FUNCTION_BLOCK SWITCHsim (* Service Interface Function Block Type *)
  (* Standard: 61499-2 *)
  (* Version 1.0, 2020-01-13, badger *)
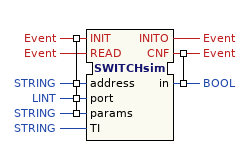
  EVENT_INPUT
    INIT WITH address, port, params; (* Initialise the switch simulator *)
    READ; (* Check the switches for changes *)
  END_EVENT
  EVENT_OUTPUT
    INITO; (* Initialisation confirmation *)
    CNF WITH in; (* Confirms that the switch has been read *)
  END_EVENT
  VAR_INPUT
    address : STRING; (* URL of the simulation server *)
    port : LINT; (* Listener port on the simulation server *)
    params : STRING; (* Zone the controller is managing and the switch being read *)
    TI : STRING; (* Requirements Traceability ID *)
  END_VAR
  VAR_OUTPUT
    in : BOOL; (* Set true if the switch was pressed or false if not. *)
  END_VAR
  SERVICE APPLICATION/RESOURCE (* Service Interface Function Block Type *)
    SEQUENCE normal_establishment
      APPLICATION.INIT+(PARAMS) -> RESOURCE.initialize(PARAMS) -> APPLICATION.INITO+();
    END_SEQUENCE
    SEQUENCE unsuccessful_establishment
      APPLICATION.INIT+(PARAMS) -> RESOURCE.initialize(PARAMS) -> APPLICATION.INITO-(STATUS);
    END_SEQUENCE
    SEQUENCE request_confirm
      APPLICATION.REQ+(SD) -> RESOURCE.request(SD) -> APPLICATION.CNF+(RD);
    END_SEQUENCE
    SEQUENCE request_inhibited
      APPLICATION.REQ-(SD) -> APPLICATION.CNF-(STATUS);
    END_SEQUENCE
    SEQUENCE request_error
      APPLICATION.REQ+(SD) -> RESOURCE.request(SD) -> APPLICATION.CNF-(STATUS);
    END_SEQUENCE
    SEQUENCE indication_response
      RESOURCE.indicate(RD) -> APPLICATION.IND+(RD);
      APPLICATION.RSP(QI,SD) -> RESOURCE.response(QI,SD);
    END_SEQUENCE
    SEQUENCE indication_inhibited
      RESOURCE.indicate(RD,QI=FALSE) -> RESOURCE.inhibited();
    END_SEQUENCE
    SEQUENCE error_indication
      RESOURCE.error(STATUS) -> APPLICATION.IND-(STATUS);
    END_SEQUENCE
    SEQUENCE application_initiated_termination
      APPLICATION.INIT-() -> RESOURCE.terminate() -> APPLICATION.INITO-(STATUS);
    END_SEQUENCE
    SEQUENCE resource_initiated_termination
      -> APPLICATION.INITO-(STATUS);
    END_SEQUENCE
  END_SERVICE
END_FUNCTION_BLOCK
